SYSTEM test
  (* Standard: 61499-1; Classification: Training; ApplicationDomain: Agriculture; Function: Learning how to use 4diac; Type: Test Type; Description: Copyright (c) 2023, 2025 HR Agrartechnik GmbH, Meisterschulen am Ostbahnhof This program and the accompanying materials are made available under the terms of the Eclipse Public License 2.0 which is available at https://www.eclipse.org/legal/epl-2.0/ SPDX-License-Identifier: EPL-2.0 https://www.logibus.tech/ Training Hier kann man über "Change Type" andere Ventilsteuerung_Uebung_001 usw auswählen, und so Übung für Übung vollziehen. Quellen: 1. Mit Musterlösungen: https://github.com/Meisterschulen-am-Ostbahnhof-Munchen/4diac_training1 2. Ohne Musterlösungen: https://github.com/Meisterschulen-am-Ostbahnhof-Munchen/4diac_training1_empty *)
  (* Version 1.0, 2025-09-28, Franz Höpfinger, HR Agrartechnik GmbH *)
  PACKAGE Training;
  IMPORT logiBUS::stations::Computers::C_00;
  APPLICATION App (* Main App for a front fertilizer *)
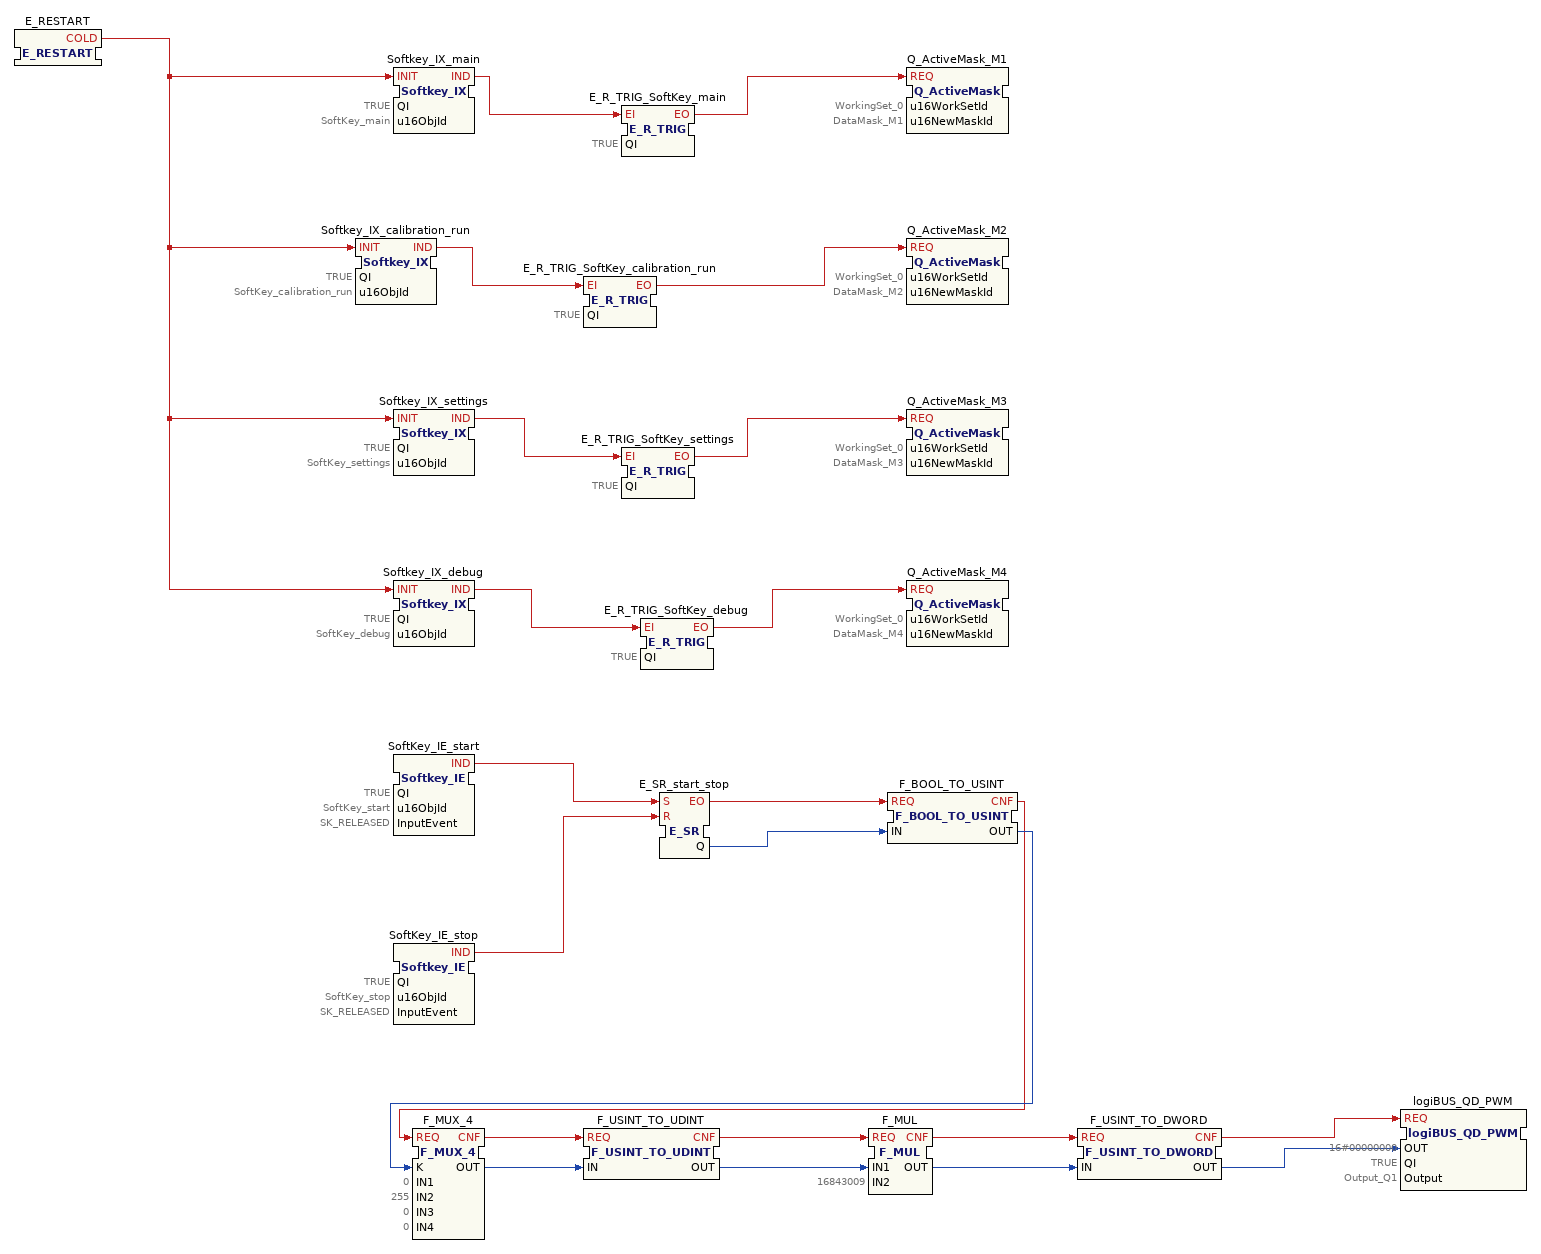
    FBS
      Softkey_IX_main : isobus::UT::io::Softkey::Softkey_IX(QI := TRUE, u16ObjId := SoftKey_main);
      Softkey_IX_calibration_run : isobus::UT::io::Softkey::Softkey_IX(QI := TRUE, u16ObjId := SoftKey_calibration_run);
      Softkey_IX_settings : isobus::UT::io::Softkey::Softkey_IX(QI := TRUE, u16ObjId := SoftKey_settings);
      Softkey_IX_debug : isobus::UT::io::Softkey::Softkey_IX(QI := TRUE, u16ObjId := SoftKey_debug);
      E_R_TRIG_SoftKey_main : iec61499::events::E_R_TRIG(QI := TRUE);
      E_R_TRIG_SoftKey_calibration_run : iec61499::events::E_R_TRIG(QI := TRUE);
      E_R_TRIG_SoftKey_settings : iec61499::events::E_R_TRIG(QI := TRUE);
      E_R_TRIG_SoftKey_debug : iec61499::events::E_R_TRIG(QI := TRUE);
      Q_ActiveMask_M1 : isobus::UT::Q::Q_ActiveMask(u16WorkSetId := WorkingSet_0, u16NewMaskId := DataMask_M1);
      Q_ActiveMask_M2 : isobus::UT::Q::Q_ActiveMask(u16WorkSetId := WorkingSet_0, u16NewMaskId := DataMask_M2);
      Q_ActiveMask_M3 : isobus::UT::Q::Q_ActiveMask(u16WorkSetId := WorkingSet_0, u16NewMaskId := DataMask_M3);
      Q_ActiveMask_M4 : isobus::UT::Q::Q_ActiveMask(u16WorkSetId := WorkingSet_0, u16NewMaskId := DataMask_M4);
      E_RESTART : iec61499::events::E_RESTART;
      SoftKey_IE_start : isobus::UT::io::Softkey::Softkey_IE(QI := TRUE, u16ObjId := SoftKey_start, InputEvent := SK_RELEASED);
      SoftKey_IE_stop : isobus::UT::io::Softkey::Softkey_IE(QI := TRUE, u16ObjId := SoftKey_stop, InputEvent := SK_RELEASED);
      E_SR_start_stop : iec61499::events::E_SR;
      logiBUS_QD_PWM : logiBUS::io::DQ::logiBUS_QD_PWM(QI := TRUE, OUT := 16#00000000, Output := Output_Q1);
      F_USINT_TO_DWORD : iec61131::conversion::F_USINT_TO_DWORD;
      F_MUL : iec61131::arithmetic::F_MUL(IN2 := 16843009);
      F_USINT_TO_UDINT : iec61131::conversion::F_USINT_TO_UDINT;
      F_MUX_4 : iec61131::selection::F_MUX_4(IN1 := 0, IN2 := 255 (* Automatic *), IN3 := 0, IN4 := 0);
      F_BOOL_TO_USINT : iec61131::conversion::F_BOOL_TO_USINT;
    END_FBS
    EVENT_CONNECTIONS
      Softkey_IX_main.IND TO E_R_TRIG_SoftKey_main.EI;
      E_R_TRIG_SoftKey_main.EO TO Q_ActiveMask_M1.REQ;
      E_RESTART.COLD TO Softkey_IX_main.INIT;
      Softkey_IX_calibration_run.IND TO E_R_TRIG_SoftKey_calibration_run.EI;
      E_R_TRIG_SoftKey_calibration_run.EO TO Q_ActiveMask_M2.REQ;
      Softkey_IX_settings.IND TO E_R_TRIG_SoftKey_settings.EI;
      Softkey_IX_debug.IND TO E_R_TRIG_SoftKey_debug.EI;
      E_R_TRIG_SoftKey_settings.EO TO Q_ActiveMask_M3.REQ;
      E_R_TRIG_SoftKey_debug.EO TO Q_ActiveMask_M4.REQ;
      E_RESTART.COLD TO Softkey_IX_calibration_run.INIT;
      E_RESTART.COLD TO Softkey_IX_settings.INIT;
      E_RESTART.COLD TO Softkey_IX_debug.INIT;
      SoftKey_IE_start.IND TO E_SR_start_stop.S;
      SoftKey_IE_stop.IND TO E_SR_start_stop.R;
      F_USINT_TO_DWORD.CNF TO logiBUS_QD_PWM.REQ;
      F_MUL.CNF TO F_USINT_TO_DWORD.REQ;
      F_USINT_TO_UDINT.CNF TO F_MUL.REQ;
      F_MUX_4.CNF TO F_USINT_TO_UDINT.REQ;
      E_SR_start_stop.EO TO F_BOOL_TO_USINT.REQ;
      F_BOOL_TO_USINT.CNF TO F_MUX_4.REQ;
    END_CONNECTIONS
    DATA_CONNECTIONS
      F_USINT_TO_DWORD.OUT TO logiBUS_QD_PWM.OUT;
      F_MUL.OUT TO F_USINT_TO_DWORD.IN;
      F_USINT_TO_UDINT.OUT TO F_MUL.IN1;
      F_MUX_4.OUT TO F_USINT_TO_UDINT.IN;
      E_SR_start_stop.Q TO F_BOOL_TO_USINT.IN;
      F_BOOL_TO_USINT.OUT TO F_MUX_4.K;
    END_CONNECTIONS
  END_APPLICATION
  DEVICE FORTE_PC : (MGR_ID := C_00 (* Device manager socket ID *))
    {SET_ATTRIBUTE(Profile, HOLOBLOC)}
    RESOURCE EMB_RES : 
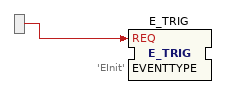
      FBS
        E_TRIG : iec61499::events::E_TRIG(EVENTTYPE := 'EInit');
      END_FBS
      EVENT_CONNECTIONS
         TO E_TRIG.REQ;
      END_CONNECTIONS
    END_RESOURCE
  END_DEVICE
END_SYSTEM
